(* IEC 61131-3 sources: STruCpp/libs/sources/additional-function-blocks, 6 files *)

(* ---- derivative.st ---- *)
(* Additional Function Blocks: DERIVATIVE                                *)
(* Source: example function block of IEC 61131-3, 2nd Ed.                *)

FUNCTION_BLOCK DERIVATIVE
  VAR_INPUT
    RUN   : BOOL ;          (* 0 = reset                  *)
    XIN   : REAL ;          (* Input to be differentiated *)
    CYCLE : TIME ;          (* Sampling period            *)
  END_VAR
  VAR_OUTPUT
    XOUT : REAL ;           (* Differentiated output      *)
  END_VAR
  VAR
    X1 : REAL ;
    X2 : REAL ;
    X3 : REAL ;
  END_VAR

  IF RUN THEN
    XOUT := (3.0 * (XIN - X3) + X1 - X2) / (10.0 * TIME_TO_REAL(CYCLE)) ;
    X3 := X2 ;
    X2 := X1 ;
    X1 := XIN ;
  ELSE
    XOUT := 0.0 ;
    X1 := XIN ;
    X2 := XIN ;
    X3 := XIN ;
  END_IF ;
END_FUNCTION_BLOCK

(* ---- hysteresis.st ---- *)
(* Additional Function Blocks: HYSTERESIS                                *)
(* Source: example function block of IEC 61131-3, 2nd Ed.                *)
(*                                                                        *)
(* Boolean hysteresis on the difference of two REAL inputs (XIN1 - XIN2). *)

FUNCTION_BLOCK HYSTERESIS
  VAR_INPUT
    XIN1 : REAL ;
    XIN2 : REAL ;
    EPS  : REAL ;
  END_VAR
  VAR_OUTPUT
    Q : BOOL := FALSE ;
  END_VAR

  IF Q THEN
    IF XIN1 < (XIN2 - EPS) THEN
      Q := FALSE ;
    END_IF ;
  ELSIF XIN1 > (XIN2 + EPS) THEN
    Q := TRUE ;
  END_IF ;
END_FUNCTION_BLOCK

(* ---- integral.st ---- *)
(* Additional Function Blocks: INTEGRAL                                  *)
(* Source: example function block of IEC 61131-3, 2nd Ed.                *)

FUNCTION_BLOCK INTEGRAL
  VAR_INPUT
    RUN   : BOOL ;       (* 1 = integrate, 0 = hold *)
    R1    : BOOL ;       (* Overriding reset        *)
    XIN   : REAL ;       (* Input variable          *)
    X0    : REAL ;       (* Initial value           *)
    CYCLE : TIME ;       (* Sampling period         *)
  END_VAR
  VAR_OUTPUT
    Q    : BOOL ;        (* NOT R1                  *)
    XOUT : REAL ;        (* Integrated output       *)
  END_VAR

  Q := NOT R1 ;
  IF R1 THEN
    XOUT := X0 ;
  ELSIF RUN THEN
    XOUT := XOUT + XIN * TIME_TO_REAL(CYCLE) ;
  END_IF ;
END_FUNCTION_BLOCK

(* ---- pid.st ---- *)
(* Additional Function Blocks: PID                                       *)
(* Source: example function block of IEC 61131-3, 2nd Ed.                *)
(*                                                                        *)
(* Depends on INTEGRAL and DERIVATIVE FBs declared elsewhere in this lib. *)

FUNCTION_BLOCK PID
  VAR_INPUT
    AUTO  : BOOL ;       (* 0 - manual , 1 - automatic *)
    PV    : REAL ;       (* Process variable *)
    SP    : REAL ;       (* Set point *)
    X0    : REAL ;       (* Manual output adjustment - typically from transfer station *)
    KP    : REAL ;       (* Proportionality constant *)
    TR    : REAL ;       (* Reset time *)
    TD    : REAL ;       (* Derivative time constant *)
    CYCLE : TIME ;       (* Sampling period *)
  END_VAR
  VAR_OUTPUT
    XOUT : REAL ;
  END_VAR
  VAR
    ERROR : REAL ;        (* PV - SP *)
    ITERM : INTEGRAL ;    (* FB for integral term  *)
    DTERM : DERIVATIVE ;  (* FB for derivative term *)
  END_VAR

  ERROR := PV - SP ;
  (*** Adjust ITERM so that XOUT := X0 when AUTO = 0 ***)
  ITERM (RUN := AUTO, R1 := NOT AUTO, XIN := ERROR,
         X0 := TR * (X0 - ERROR), CYCLE := CYCLE) ;
  DTERM (RUN := AUTO, XIN := ERROR, CYCLE := CYCLE) ;
  XOUT := KP * (ERROR + ITERM.XOUT / TR + DTERM.XOUT * TD) ;
END_FUNCTION_BLOCK

(* ---- ramp.st ---- *)
(* Additional Function Blocks: RAMP                                      *)
(* Source: example function block of IEC 61131-3, 2nd Ed.                *)

FUNCTION_BLOCK RAMP
  VAR_INPUT
    RUN   : BOOL ;       (* 0 - track X0, 1 - ramp to/track X1 *)
    X0    : REAL ;
    X1    : REAL ;
    TR    : TIME ;       (* Ramp duration *)
    CYCLE : TIME ;       (* Sampling period *)
  END_VAR
  VAR_OUTPUT
    BUSY : BOOL ;        (* BUSY = 1 during ramping period *)
    XOUT : REAL := 0.0 ;
  END_VAR
  VAR
    XI : REAL ;          (* Initial value *)
    T  : TIME := T#0s ;  (* Elapsed time of ramp *)
  END_VAR

  BUSY := RUN ;
  IF RUN THEN
    IF T >= TR THEN
      BUSY := FALSE ;
      XOUT := X1 ;
    ELSE
      XOUT := XI + (X1 - XI) * TIME_TO_REAL(T) / TIME_TO_REAL(TR) ;
      T := T + CYCLE ;
    END_IF ;
  ELSE
    XOUT := X0 ;
    XI := X0 ;
    T := T#0s ;
  END_IF ;
END_FUNCTION_BLOCK

(* ---- rtc.st ---- *)
(* SPDX-License-Identifier: GPL-3.0-only WITH STruCpp-runtime-exception *)
(* Copyright (c) 2026 Autonomy® *)
(* Additional Function Blocks: RTC (real time clock)                      *)
(* First scan: CDT starts from CURRENT_DT() (1970 + uptime on targets     *)
(* without a system date). SET = TRUE: CDT = PDT. SET = FALSE: CDT counts *)
(* on from the last start value. Q copies SET.                            *)

FUNCTION_BLOCK RTC
  VAR_INPUT
    SET : BOOL ;
    PDT : DT ;
  END_VAR
  VAR_OUTPUT
    Q   : BOOL := FALSE ;
    CDT : DT ;
  END_VAR
  VAR
    started  : BOOL := FALSE ;
    preset   : DT ;
    set_time : TIME ;
  END_VAR

  IF SET THEN
    preset := PDT ;
    set_time := TIME() ;
    started := TRUE ;
  ELSIF NOT started THEN
    preset := CURRENT_DT() ;
    set_time := TIME() ;
    started := TRUE ;
  END_IF ;
  CDT := preset + (TIME() - set_time) ;
  Q := SET ;
END_FUNCTION_BLOCK
